// folder: (top level)

FUNCTION_BLOCK "Block_1"   // FB1, SCL
{ S7_Optimized_Access := 'TRUE' }
VERSION : 0.1
BEGIN

   IF "DB_State".State = "CHECK" THEN
       IF "MagE_D" = TRUE THEN
           "MCDIR" := 0;
           "DB_State".State := "START";
       ELSE
           "MCDIR" := 1;
           "DB_State".State := "INIT";
       END_IF;

   ELSIF "DB_State".State = "INIT" THEN
       "MCDIR" := 1;
       IF "MagE_D" = TRUE THEN
           "MCDIR" := 0;
           "DB_State".State := "CHECK";

       END_IF;

   ELSIF "DB_State".State = "START" THEN 
       "MCDIR" := 1;
       IF "IndNS_SS" = TRUE OR "IndNS_SS" = TRUE OR "IndNS_SS" = TRUE THEN
           "MCDIR" := 0;
           "DB_State".State := "PROCESS";
       END_IF;

   ELSIF "DB_State".State = "PROCESS" THEN //
       "MCDIR" := 0;
       "ZendDO" := TRUE;
       "ZendUP" := FALSE;
       // Start the timer if it is not running
       IF "DB_State".TimerFlag = FALSE THEN
           "Timer_Cylinder".TON(IN:=TRUE,
                                PT:=T#4s,
                                Q=>"DB_State".TimerFlag);
       END_IF;

       // Check if the timer has elapsed
       IF "DB_State".TimerFlag  THEN
           "ZendUP" := TRUE; 
           "ZendDO" := FALSE;
       END_IF;

       "DB_State".State := "START";


   END_IF;
END_FUNCTION_BLOCK

FUNCTION "Bsp3.1" : Void   // FC1, SCL
{ S7_Optimized_Access := 'TRUE' }
VERSION : 0.1
BEGIN
   IF "Swt0-7" <= 27 THEN
       "LED0-7" := "Swt0-7";
       ;
   ELSE
       "LED0-7" := 0;
   END_IF;
END_FUNCTION

FUNCTION "Bsp3.2" : Void   // FC2, SCL
{ S7_Optimized_Access := 'TRUE' }
VERSION : 0.1
BEGIN

   "Lampe_0" := "Clock_1Hz";
END_FUNCTION

FUNCTION "Bsp3.2_mit_timer" : Void   // FC3, SCL
{ S7_Optimized_Access := 'TRUE' }
VERSION : 0.1
BEGIN
   "Timer_3.2".TP(IN:="Clock_1Hz",
                  PT:=T#250ms,
                  Q=>"Lampe_0");
END_FUNCTION

FUNCTION "Bsp3.3" : Void   // FC4, SCL
{ S7_Optimized_Access := 'TRUE' }
VERSION : 0.1
   VAR CONSTANT
      JOY_MAX : Int := 1500;
      JOY_MIN : Int := -1500;
      JOY_MITTE : Int := 50;
   END_VAR
BEGIN
   IF "JOY_LeftRight" < 0.9 * #JOY_MIN THEN
       "LED3" := FALSE;
       "LED4" := FALSE;
       "LED5" := FALSE;
       "LED6" := TRUE;
   ELSIF "JOY_LeftRight" < 0.6 * #JOY_MIN THEN
       "LED3" := FALSE;
       "LED4" := FALSE;
       "LED5" := TRUE;
       "LED6" := FALSE;
   ELSIF "JOY_LeftRight" < 0.3 * #JOY_MIN THEN
       "LED3" := FALSE;
       "LED4" := TRUE;
       "LED5" := FALSE;
       "LED6" := FALSE;
   ELSIF "JOY_LeftRight" >= 0.3 * #JOY_MIN AND "JOY_LeftRight" <= #JOY_MITTE THEN
       "LED3" := TRUE;
       "LED4" := FALSE;
       "LED5" := FALSE;
       "LED6" := FALSE;
   ELSE
       "LED3" := FALSE;
       "LED4" := FALSE;
       "LED5" := FALSE;
       "LED6" := FALSE;
   END_IF;
END_FUNCTION

FUNCTION "Bsp3.4" : Void   // FC5, SCL
{ S7_Optimized_Access := 'TRUE' }
VERSION : 0.1
   VAR CONSTANT
      INT_MAX : Int := 16#FFFF;
   END_VAR
BEGIN
   //"MCSPEED" := #INT_MAX

   IF "DB_State".State = 0 THEN
       IF "MagE_D" = TRUE THEN
           "MCDIR" := 0;
           "DB_State".State := 1;
       ELSE
           "MCDIR" := 1;
           "DB_State".State := 2;
       END_IF;

   ELSIF "DB_State".State = 1 THEN
       "MCDIR" := 0;
       IF "MagE_U" = TRUE THEN
           "MCDIR" := 1;
           "DB_State".State := 2;

       END_IF;

   ELSIF "DB_State".State = 2 THEN
       "MCDIR" := 1;
       IF "MagE_D" = TRUE THEN
           "MCDIR" := 0;
           "DB_State".State := 1;

       END_IF;
   END_IF;

   IF "Swt7" THEN
       "MCGO" := TRUE;
       "Lampe_1" := FALSE;
       "Lampe_2" := TRUE;
      /// "DB_State".State := 0;
   ELSE
       "Lampe_1" := TRUE;
       "Lampe_2" := FALSE;
       "MCGO" := FALSE;
       //"DB_State".State := 10;
   END_IF;
END_FUNCTION

ORGANIZATION_BLOCK "Main"   // OB1, SCL, ProgramCycle
TITLE = "Main Program Sweep (Cycle)"
{ S7_Optimized_Access := 'TRUE' }
VERSION : 0.1
BEGIN

   "Block_1_DB"();
END_ORGANIZATION_BLOCK

// ===== PLC "Target_2"  CPU 1214C DC/DC/DC =====

VAR_GLOBAL   // PLC tag table "Standard-Variablentabelle"
   "Clock_2.5Hz" AT %M8000.2 : Bool;
   "Clock_2Hz" AT %M8000.3 : Bool;
   "Clock_1.25Hz" AT %M8000.4 : Bool;
   "Clock_1Hz" AT %M8000.5 : Bool;
   "Clock_0.625Hz" AT %M8000.6 : Bool;
   "Clock_0.5Hz" AT %M8000.7 : Bool;
   "System_Byte" AT %MB8001 : Byte;
   "FirstScan" AT %M8001.0 : Bool;
   "AlwaysTRUE" AT %M8001.2 : Bool;
   "AlwaysFALSE" AT %M8001.3 : Bool;
END_VAR

ORGANIZATION_BLOCK "Main"   // OB1, LAD, ProgramCycle
TITLE = "Main Program Sweep (Cycle)"
{ S7_Optimized_Access := 'TRUE' }
VERSION : 0.1
BEGIN
END_ORGANIZATION_BLOCK

(* ===== HMI "HMI_RT_1" =====
system functions are stored by id; their names below are inferred from use
connection "HMI_Connection_1": ETHERNET, S7_1200_OMS

HMI tags "Default tag table"
   "Tag_ScreenNumber" : UInt, internal

text list "Textliste_Bildnamen": 1 'Root screen'

screen "Root screen" 480x212, template "Template_1"
   on GenerateScreen: SetTag("Tag_ScreenNumber", 1)
   TextField "HmiScreenItemData" at 48,60 size 384x22; Text 'Willkommen zum HMI_1 (KTP400 Comfort)!'

Template "Template_1" 480x212
   Button "Beenden" at 379,148 size 63x63; TextOff 'Beenden'; PictureOff "ExitRuntime_KTP400_Comfort_TR"; PictureOn "ExitRuntime_KTP400_Comfort_TR"
      on Release: StopRuntime(0)
   Button "Template_Button" at 265,148 size 63x63; TextOff 'Text'
   Button "Meldungen" at 151,148 size 63x63; TextOff 'Meldungen'; PictureOff "AlarmDisplay_KTP400_Comfort_TR"; PictureOn "AlarmDisplay_KTP400_Comfort_TR"
      on Release: function_ef3f5d25("Alarm window_Unacknowledged", -1)
   Button "Startbild" at 37,148 size 63x63; TextOff 'Startbild'; PictureOff "NavigateHome_KTP400_Comfort_TR"; PictureOn "NavigateHome_KTP400_Comfort_TR"
      on Release: ActivateScreen("Root screen", 0)
*)

(* ===== HMI "HMI_RT_2" =====
system functions are stored by id; their names below are inferred from use
connection "HMI_Connection_2": ETHERNET, S7_1200_OMS

HMI tags "Default tag table"
   "Tag_ScreenNumber" : UInt, internal

text list "Textliste_Bildnamen": 1 'Root screen'

screen "Root screen" 480x212, template "Template_1"
   on GenerateScreen: SetTag("Tag_ScreenNumber", 1)
   TextField "HmiScreenItemData" at 48,60 size 384x22; Text 'Willkommen zum HMI_2 (KTP400 Comfort)!'

Template "Template_1" 480x212
   Button "Beenden" at 379,148 size 63x63; TextOn 'Beenden'; TextOff 'Beenden'; PictureOn "ExitRuntime_KTP400_Comfort_TR"; PictureOff "ExitRuntime_KTP400_Comfort_TR"
      on Release: StopRuntime(0)
   Button "Template_Button" at 265,148 size 63x63; TextOff 'Text'
   Button "Meldungen" at 151,148 size 63x63; TextOn 'Meldungen'; TextOff 'Meldungen'; PictureOn "AlarmDisplay_KTP400_Comfort_TR"; PictureOff "AlarmDisplay_KTP400_Comfort_TR"
      on Release: function_ef3f5d25("Alarm window_Unacknowledged", -1)
   Button "Startbild" at 37,148 size 63x63; TextOn 'Startbild'; TextOff 'Startbild'; PictureOn "NavigateHome_KTP400_Comfort_TR"; PictureOff "NavigateHome_KTP400_Comfort_TR"
      on Release: ActivateScreen("Root screen", 0)
*)

(* ===== HMI "HMI_RT_3" =====
system functions are stored by id; their names below are inferred from use
connection "HMI_Connection_3": ETHERNET, S7_1200_OMS

HMI tags "Default tag table"
   "Tag_ScreenNumber" : UInt, internal

text list "Textliste_Bildnamen": 1 'Root screen'

screen "Root screen" 480x212, template "Template_1"
   on GenerateScreen: SetTag("Tag_ScreenNumber", 1)
   TextField "HmiScreenItemData" at 48,60 size 384x22; Text 'Willkommen zum HMI_3 (KTP400 Comfort)!'

Template "Template_1" 480x212
   Button "Beenden" at 379,148 size 63x63; TextOn 'Beenden'; TextOff 'Beenden'; PictureOn "ExitRuntime_KTP400_Comfort_TR"; PictureOff "ExitRuntime_KTP400_Comfort_TR"
      on Release: StopRuntime(0)
   Button "Template_Button" at 265,148 size 63x63; TextOff 'Text'
   Button "Meldungen" at 151,148 size 63x63; TextOn 'Meldungen'; TextOff 'Meldungen'; PictureOn "AlarmDisplay_KTP400_Comfort_TR"; PictureOff "AlarmDisplay_KTP400_Comfort_TR"
      on Release: function_ef3f5d25("Alarm window_Unacknowledged", -1)
   Button "Startbild" at 37,148 size 63x63; TextOn 'Startbild'; TextOff 'Startbild'; PictureOn "NavigateHome_KTP400_Comfort_TR"; PictureOff "NavigateHome_KTP400_Comfort_TR"
      on Release: ActivateScreen("Root screen", 0)
*)

(* ===== HMI "HMI_RT_4" =====
system functions are stored by id; their names below are inferred from use
connection "HMI_Connection_4": ETHERNET, S7_1200_OMS

HMI tags "Default tag table"
   "Tag_ScreenNumber" : UInt, internal

text list "Textliste_Bildnamen": 1 'Root screen'

screen "Root screen" 480x212, template "Template_1"
   on GenerateScreen: SetTag("Tag_ScreenNumber", 1)
   TextField "HmiScreenItemData" at 48,60 size 384x22; Text 'Willkommen zum HMI_4 (KTP400 Comfort)!'

Template "Template_1" 480x212
   Button "Beenden" at 379,148 size 63x63; TextOn 'Beenden'; TextOff 'Beenden'; PictureOn "ExitRuntime_KTP400_Comfort_TR"; PictureOff "ExitRuntime_KTP400_Comfort_TR"
      on Release: StopRuntime(0)
   Button "Template_Button" at 265,148 size 63x63; TextOff 'Text'
   Button "Meldungen" at 151,148 size 63x63; TextOn 'Meldungen'; TextOff 'Meldungen'; PictureOn "AlarmDisplay_KTP400_Comfort_TR"; PictureOff "AlarmDisplay_KTP400_Comfort_TR"
      on Release: function_ef3f5d25("Alarm window_Unacknowledged", -1)
   Button "Startbild" at 37,148 size 63x63; TextOn 'Startbild'; TextOff 'Startbild'; PictureOn "NavigateHome_KTP400_Comfort_TR"; PictureOff "NavigateHome_KTP400_Comfort_TR"
      on Release: ActivateScreen("Root screen", 0)
*)

(* ===== HMI "HMI_RT_5" =====
system functions are stored by id; their names below are inferred from use
connection "HMI_Connection_5": ETHERNET, S7_1200_OMS

HMI tags "Default tag table"
   "Tag_ScreenNumber" : UInt, internal
   "State" : UInt = PLC DB_State.State, 1 s
   "Tank" : Int = PLC Block_1_DB.tank AT %DB1.DBW0, 1 s
   "KapNs" : Bool = PLC Block_1_DB.CapSen AT %DB1.DBW0, 1 s
   "ElMag" : Bool = PLC Block_1_DB.MagSen AT %DB1.DBW0, 1 s
   "IndNS" : Bool = PLC Block_1_DB.IndSen AT %DB1.DBW0, 1 s
   "OptNS" : Bool = PLC Block_1_DB.OptSen AT %DB1.DBW0, 1 s
   "NumPieces" : Int = PLC Block_1_DB.NumPieces AT %DB1.DBW0, 1 s
   "MCGO" : Bool = PLC MCGO AT %Q5.2, 1 s
   "MCDIR" : Bool = PLC MCDIR AT %Q5.3, 1 s
   "ZylUp" : Bool = PLC ZylUp AT %Q8.3, 1 s
   "ZylDown" : Bool = PLC ZylDown AT %Q8.2, 1 s
   "JoyUpDown" : Int = PLC JOY_UpDown AT %IW68, 1 s
   "Prev_State" : UInt = PLC Block_1_DB.Prev_State AT %DB1.DBW0, 1 s
   "Man_Mode" : Bool = PLC Block_1_DB.Man_Mode AT %DB1.DBX0.0, 1 s
   "Cyl_Down" : Bool = PLC Block_1_DB.Cyl_Down AT %DB1.DBX0.0, 1 s
   "Man_Move" : Int = PLC Block_1_DB.Man_Move AT %DB1.DBX0.0, 1 s
   "Errors" : Word = PLC Block_1_DB.Errors AT %DB1.DBW0, 1 s
   "Temp" : Int = PLC Block_1_DB.temp AT %DB14.DBB2, 1 s

discrete alarms
   1: 'Error: Person in tank vicinity', class Errors, trigger "Errors" bit 3
   2: 'Error: No piece in trolley', class Errors, trigger "Errors" bit 1
   3: 'Error: Sensor could be damaged!', class Errors, trigger "Errors" bit 2
   4: 'Warning: Tank Placed Incorrectly', class Warnings, trigger "Errors" bit 4
   5: 'Info: Test Run in progress!', class Acknowledgement, trigger "Errors" bit 5
   6: 'Info: Normal Run in progress', class Acknowledgement, trigger "Errors" bit 6
   7: 'Warning: Too Hot!', class Warnings, trigger "Errors" bit 7

text list "Textliste_Bildnamen": 1 'Root screen'

screen "Root" 480x272, template "Template_1"
   on GenerateScreen: SetTag("Tag_ScreenNumber", 1)
   Button "Button_1" at 38,35 size 71x53; TextOff 'Viz'
      on Press: ActivateScreen("Visualisation", 0)
   Button "Button_2" at 202,35 size 71x53; TextOff 'Log'
      on Press: ActivateScreen("Log", 0)
   Button "Button_3" at 366,35 size 71x53; TextOff 'Man'
      on Click: ActivateScreen("Manual", 0)

Template "Template_1" 480x272
   Button "Beenden" at 379,148 size 63x63; TextOn 'Beenden'; TextOff 'Beenden'; PictureOn "ExitRuntime_KTP400_Comfort_TR"; PictureOff "ExitRuntime_KTP400_Comfort_TR"
      on Release: StopRuntime(0)
   Button "Template_Button" at 265,148 size 63x63; TextOff 'Text'
   Button "Meldungen" at 151,148 size 63x63; TextOn 'Meldungen'; TextOff 'Meldungen'; PictureOn "AlarmDisplay_KTP400_Comfort_TR"; PictureOff "AlarmDisplay_KTP400_Comfort_TR"
      on Release: function_ef3f5d25("Alarm window_Unacknowledged", -1)
   Button "Startbild" at 37,148 size 63x63; TextOn 'Startbild'; TextOff 'Startbild'; PictureOn "NavigateHome_KTP400_Comfort_TR"; PictureOff "NavigateHome_KTP400_Comfort_TR"
      on Release: ActivateScreen("Root", 0)

screen "Log" 480x272
   TextField "Text field_5" at 373,11 size 107x20; Text 'Num of Pieces'
   IOField "I/O field_1" at 424,56 size 41x32; FormatPattern 99
      ProcessValue <- "NumPieces"
   Button "Button_1" at 404,207 size 74x53; TextOff 'Text'; PictureOff "Home"
      on Click: ActivateScreen("Root", 0)
   AlarmView "Alarm view_1" at 11,7 size 354x190
   Circle "Circle_4" at 129,219 size 53x53
      Appearance <- "OptNS"
   TextField "Text field_1" at 31,199 size 47x20; Text 'IndNS'
   Circle "Circle_1" at 25,219 size 53x53
      Appearance <- "IndNS"
   TextField "Text field_2" at 137,199 size 50x20; Text 'KapNS'
   Circle "Circle_2" at 228,219 size 53x53
      Appearance <- "KapNs"
   TextField "Text field_3" at 236,197 size 47x20; Text 'ElMag'
   Circle "Circle_3" at 320,219 size 53x53
      Appearance <- "ElMag"
   TextField "Text field_4" at 326,199 size 49x20; Text 'OptNS'

screen "Visualisation" 480x272
   TextField "Text field_1" at 9,29 size 219x20; Text 'Trolley currently at station:'
   TextField "Text field_2" at 221,29 size 14x20; Text 'Text'
   Slider "Slider_1" at 52,60 size 71x110; Caption 'SIMATIC'
      ProcessValue <- "Tank"
   TextField "Text field_3" at 62,186 size 43x20; Text 'Error'
   TextField "Text field_4" at 246,32 size 197x20; Text 'Is piece being processed?'
   Circle "Circle_1" at 309,65 size 39x39
      Appearance <- "State"
   Button "Button_1" at 35,206 size 96x51; TextOff 'Error'; PictureOff "Graphic_2"
      Appearance <- "State"
      on Click: SetTag("State", 9); SetTag("Errors", 0)
   Button "Button_2" at 404,157 size 74x53; TextOff 'Text'; PictureOff "Home"
      on Click: ActivateScreen("Root", 0)
   Bar "Bar_1" at 207,107 size 55x126; MinimumValue 0; MaximumValue 100
      ProcessValue <- "Temp"
   TextField "Text field_5" at 194,240 size 100x20; Text 'Temperature'

screen "Manual" 480x272
   Button "Button_1" at 53,122 size 110x72; TextOff 'Down'
      on Press: SetTag("Man_Move", -1)
      on Release: SetTag("Man_Move", 0)
   Switch "Switch_2" at 228,104 size 157x90; CaptionText 'Cylinder'; TextOff 'Down'; TextOn 'Up'
      on SwitchOn: SetTag("Cyl_Down", 1)
      on SwitchOff: SetTag("Cyl_Down", 0)
   Button "Button_2" at 404,157 size 74x53; TextOff 'Text'; PictureOff "Home"
      on Click: ActivateScreen("Root", 0)
   Switch "Switch_3" at 228,6 size 161x85; CaptionText 'Manual Mode'; TextOff 'OFF'; TextOn 'ON'
      on SwitchOn: SetTag("Man_Mode", 1)
      on SwitchOff: SetTag("Man_Mode", 0)
      ProcessValue <- "Man_Mode"
   Button "Button_3" at 53,19 size 110x72; TextOff 'Up'
      on Press: SetTag("Man_Move", 1)
      on Release: SetTag("Man_Move", 0)
*)